FUNCTION_BLOCK FB_Con_2_Value
VAR_INPUT
	iInput			:	INT;
	
	tRefresh		:	TIME;
	
	diUpperMax		:	DINT	:= 32767;
	diLowerMin		:	DINT	:= 0;
	diUppMeasureVal	:	DINT;
	diLowMeasureVal	:	DINT;

	iResultMulti	:	INT		:= 1;
END_VAR
VAR_OUTPUT
	diOut			:	DINT;
END_VAR
VAR
	rX				:	REAL;
	tonBlock		:	TON;
	
	bInit			:	BOOL := FALSE;
	
	rValuePerStep	:	REAL;
END_VAR

//Blocker for refresh interval
tonBlock(IN := NOT tonBlock.Q, PT := tRefresh);

IF NOT bInit THEN
	//Calculate inital Step Size
	rValuePerStep	:= ( (DINT_TO_REAL(diUppMeasureVal + (diLowMeasureVal * (-1)))) / DINT_TO_REAL(32767));
	bInit := TRUE;
END_IF

IF tonBlock.Q THEN
	//Check for Value to set for Max Output
	IF (iInput < diLowerMin) THEN
		rX := DINT_TO_REAL(diLowMeasureVal);

	//Check for Value to set for Min Output
	ELSIF (iInput > diUpperMax) THEN
		rx := DINT_TO_REAL(diUppMeasureVal);

	//Regular calculation
	ELSE
		rX := iInput * rValuePerStep;
		
		//Reduce to minus value if needed
		IF diLowMeasureVal < 0 THEN
		
			rX := rX + DINT_TO_REAL(diLowMeasureVal);
			// plus bec. values is MNUS
		
		END_IF
	END_IF
	
	IF rX > DINT_TO_REAL(diUppMeasureVal) THEN
	
		rX := DINT_TO_REAL(diUppMeasureVal);
	
	ELSIF rX < DINT_TO_REAL(diLowMeasureVal) THEN
		
		rX := DINT_TO_REAL(diLowMeasureVal);
		
	END_IF
	
	diOut := REAL_TO_DINT(rX * iResultMulti);
	

	
END_IF

END_FUNCTION_BLOCK

(* stored: Version 1.1.0.1, ProductVersion 3.1.4024.13
   POU FB_Con_2_Value: Id {489a1907-e1bb-4e3d-874c-4a0de1eeb1d8}, SpecialFunc None *)
